TYPE DigitalOutputBase_1FE0D5EE :
STRUCT
END_STRUCT
END_TYPE

(* stored: Version 1.2.0.0, ProductVersion 3.1.4024.9
   DUT DigitalOutputBase_1FE0D5EE: Id {ac709c49-a324-4ac7-8d4f-8891b5d86cc1} *)
